// TwinCAT 3 PLC project Main
// Title: nepionic-packml
// Company: nepionic
// ProjectVersion: 0.1.0
// ProgramVersion: 3.1.4026.1+c9eadab3edd020c56c333d811d5b3c408c2550c8
// project tree:
//   Commands/ I_AbortedCommands.TcIO, I_AbortingCommands.TcIO, I_ClearingCommands.TcIO, I_CompleteCommands.TcIO, I_CompletingCommands.TcIO, I_ExecuteCommands.TcIO, I_HeldCommands.TcIO, I_HoldingCommands.TcIO, I_IdleCommands.TcIO, I_ResettingCommands.TcIO, I_StartingCommands.TcIO, I_StoppedCommands.TcIO, I_StoppingCommands.TcIO, I_SuspendedCommands.TcIO, I_SuspendingCommands.TcIO, I_UnholdingCommands.TcIO, I_UnsuspendingCommands.TcIO
//   StateMachine/ State.TcDUT, StateMachine.TcPOU
//   UnitMode/ I_UnitMode.TcIO, UnitMode.TcPOU

// ---- StateMachine/State.TcDUT
{attribute 'qualified_only'}
{attribute 'strict'}
TYPE State :
(
	UNDEFINED := 0,
    CLEARING := 1,
    STOPPED := 2,
    STARTING := 3,
    IDLE := 4,
    SUSPENDED := 5,
	EXECUTE := 6,
    STOPPING := 7,
    ABORTING := 8,
    ABORTED := 9,
    HOLDING := 10,
    HELD := 11,
    UNHOLDING := 12,
    SUSPENDING := 13,
    UNSUSPENDING := 14,
    RESETTING := 15,
    COMPLETING := 16,
    COMPLETE := 17
);
END_TYPE

// ---- Commands/I_AbortedCommands.TcIO
INTERFACE PUBLIC I_AbortedCommands

METHOD PUBLIC Clear
END_METHOD

END_INTERFACE

// ---- Commands/I_AbortingCommands.TcIO
INTERFACE PUBLIC I_AbortingCommands

METHOD PUBLIC StateComplete
END_METHOD

END_INTERFACE

// ---- Commands/I_ClearingCommands.TcIO
INTERFACE PUBLIC I_ClearingCommands

METHOD PUBLIC Abort
END_METHOD

METHOD PUBLIC StateComplete
END_METHOD

END_INTERFACE

// ---- Commands/I_CompleteCommands.TcIO
INTERFACE PUBLIC I_CompleteCommands

METHOD PUBLIC Abort
END_METHOD

METHOD PUBLIC Reset
END_METHOD

METHOD PUBLIC Stop
END_METHOD

END_INTERFACE

// ---- Commands/I_CompletingCommands.TcIO
INTERFACE PUBLIC I_CompletingCommands

METHOD PUBLIC Abort
END_METHOD

METHOD PUBLIC StateComplete
END_METHOD

METHOD PUBLIC Stop
END_METHOD

END_INTERFACE

// ---- Commands/I_ExecuteCommands.TcIO
INTERFACE PUBLIC I_ExecuteCommands

METHOD PUBLIC Abort
END_METHOD

METHOD PUBLIC Hold
END_METHOD

METHOD PUBLIC StateComplete
END_METHOD

METHOD PUBLIC Stop
END_METHOD

METHOD PUBLIC Suspend
END_METHOD

END_INTERFACE

// ---- Commands/I_HeldCommands.TcIO
INTERFACE PUBLIC I_HeldCommands

METHOD PUBLIC Abort
END_METHOD

METHOD PUBLIC Stop
END_METHOD

METHOD PUBLIC Unhold
END_METHOD

END_INTERFACE

// ---- Commands/I_HoldingCommands.TcIO
INTERFACE PUBLIC I_HoldingCommands

METHOD PUBLIC Abort
END_METHOD

METHOD PUBLIC StateComplete
END_METHOD

METHOD PUBLIC Stop
END_METHOD

END_INTERFACE

// ---- Commands/I_IdleCommands.TcIO
INTERFACE PUBLIC I_IdleCommands

METHOD PUBLIC Abort
END_METHOD

METHOD PUBLIC Start
END_METHOD

METHOD PUBLIC Stop
END_METHOD

END_INTERFACE

// ---- Commands/I_ResettingCommands.TcIO
INTERFACE PUBLIC I_ResettingCommands

METHOD PUBLIC Abort
END_METHOD

METHOD PUBLIC StateComplete
END_METHOD

METHOD PUBLIC Stop
END_METHOD

END_INTERFACE

// ---- Commands/I_StartingCommands.TcIO
INTERFACE PUBLIC I_StartingCommands

METHOD PUBLIC Abort
END_METHOD

METHOD PUBLIC StateComplete
END_METHOD

END_INTERFACE

// ---- Commands/I_StoppedCommands.TcIO
INTERFACE I_StoppedCommands

METHOD PUBLIC Reset
END_METHOD

END_INTERFACE

// ---- Commands/I_StoppingCommands.TcIO
INTERFACE PUBLIC I_StoppingCommands

METHOD PUBLIC StateComplete
END_METHOD

END_INTERFACE

// ---- Commands/I_SuspendedCommands.TcIO
INTERFACE PUBLIC I_SuspendedCommands

METHOD PUBLIC Abort
END_METHOD

METHOD PUBLIC Stop
END_METHOD

METHOD PUBLIC Unsuspend
END_METHOD

END_INTERFACE

// ---- Commands/I_SuspendingCommands.TcIO
INTERFACE PUBLIC I_SuspendingCommands

METHOD PUBLIC Abort
END_METHOD

METHOD PUBLIC StateComplete
END_METHOD

METHOD PUBLIC Stop
END_METHOD

END_INTERFACE

// ---- Commands/I_UnholdingCommands.TcIO
INTERFACE PUBLIC I_UnholdingCommands

METHOD PUBLIC Abort
END_METHOD

METHOD PUBLIC StateComplete
END_METHOD

METHOD PUBLIC Stop
END_METHOD

END_INTERFACE

// ---- Commands/I_UnsuspendingCommands.TcIO
INTERFACE PUBLIC I_UnsuspendingCommands

METHOD PUBLIC Abort
END_METHOD

METHOD PUBLIC StateComplete
END_METHOD

METHOD PUBLIC Stop
END_METHOD

END_INTERFACE

// ---- UnitMode/I_UnitMode.TcIO
INTERFACE PUBLIC I_UnitMode

METHOD PUBLIC Abort
END_METHOD

METHOD PUBLIC Clear
END_METHOD

{attribute 'monitoring':='call'}
PROPERTY PUBLIC CurrentState : State
GET
END_GET
END_PROPERTY

METHOD PUBLIC CyclicCall
END_METHOD

METHOD PUBLIC Hold
END_METHOD

{attribute 'monitoring':='call'}
PROPERTY PUBLIC IsAborted : BOOL
GET
END_GET
END_PROPERTY

{attribute 'monitoring':='call'}
PROPERTY PUBLIC IsAborting : BOOL
GET
END_GET
END_PROPERTY

{attribute 'monitoring':='call'}
PROPERTY PUBLIC IsClearing : BOOL
GET
END_GET
END_PROPERTY

{attribute 'monitoring':='call'}
PROPERTY PUBLIC IsComplete : BOOL
GET
END_GET
END_PROPERTY

{attribute 'monitoring':='call'}
PROPERTY PUBLIC IsCompleting : BOOL
GET
END_GET
END_PROPERTY

{attribute 'monitoring':='call'}
PROPERTY PUBLIC IsExecuting : BOOL
GET
END_GET
END_PROPERTY

{attribute 'monitoring':='call'}
PROPERTY PUBLIC IsHeld : BOOL
GET
END_GET
END_PROPERTY

{attribute 'monitoring':='call'}
PROPERTY PUBLIC IsHolding : BOOL
GET
END_GET
END_PROPERTY

{attribute 'monitoring':='call'}
PROPERTY PUBLIC IsIdle : BOOL
GET
END_GET
END_PROPERTY

{attribute 'monitoring':='call'}
PROPERTY PUBLIC IsResetting : BOOL
GET
END_GET
END_PROPERTY

{attribute 'monitoring':='call'}
PROPERTY PUBLIC IsStarting : BOOL
GET
END_GET
END_PROPERTY

{attribute 'monitoring':='call'}
PROPERTY PUBLIC IsStopped : BOOL
GET
END_GET
END_PROPERTY

{attribute 'monitoring':='call'}
PROPERTY PUBLIC IsStopping : BOOL
GET
END_GET
END_PROPERTY

{attribute 'monitoring':='call'}
PROPERTY PUBLIC IsSuspended : BOOL
GET
END_GET
END_PROPERTY

{attribute 'monitoring':='call'}
PROPERTY PUBLIC IsSuspending : BOOL
GET
END_GET
END_PROPERTY

{attribute 'monitoring':='call'}
PROPERTY PUBLIC IsUnholding : BOOL
GET
END_GET
END_PROPERTY

{attribute 'monitoring':='call'}
PROPERTY PUBLIC IsUnsuspending : BOOL
GET
END_GET
END_PROPERTY

METHOD PUBLIC Reset
END_METHOD

METHOD PUBLIC Start
END_METHOD

METHOD PUBLIC Stop
END_METHOD

METHOD PUBLIC Suspend
END_METHOD

METHOD PUBLIC Unhold
END_METHOD

METHOD PUBLIC Unsuspend
END_METHOD

END_INTERFACE

// ---- StateMachine/StateMachine.TcPOU
{attribute 'linkalways'} 
{attribute 'no_explicit_call' := 'This FB is a CLASS and must be accessed using methods or properties'}
{attribute 'enable_dynamic_creation'}
FUNCTION_BLOCK PUBLIC StateMachine
IMPLEMENTS
	I_AbortingCommands,
	I_ClearingCommands,
	I_HeldCommands,
	I_CompletingCommands,
	I_ExecuteCommands,
	I_AbortedCommands,
	I_CompleteCommands,
	I_HoldingCommands,
	I_UnsuspendingCommands,
	I_UnholdingCommands,
	I_SuspendingCommands,
	I_SuspendedCommands,
	I_IdleCommands,
	I_ResettingCommands,
	I_StartingCommands,
	I_StoppedCommands,
	I_StoppingCommands
VAR
	_state : State := State.IDLE;
END_VAR

METHOD PUBLIC Abort
IF IsAborting OR IsAborted THEN
	RETURN;
END_IF

_state := State.ABORTING;
END_METHOD

METHOD PUBLIC Clear
IF IsAborted THEN 
	_state := State.CLEARING;
END_IF
END_METHOD

{attribute 'monitoring':='call'}
PROPERTY PUBLIC CurrentState : State
GET
CurrentState := _state;
END_GET
END_PROPERTY

METHOD PUBLIC Hold
IF IsExecuting THEN 
	_state := State.HOLDING;
END_IF
END_METHOD

{attribute 'monitoring':='call'}
PROPERTY PUBLIC IsAborted : BOOL
GET
IsAborted := (_state = State.ABORTED);
END_GET
END_PROPERTY

{attribute 'monitoring':='call'}
PROPERTY PUBLIC IsAborting : BOOL
GET
IsAborting := (_state = State.ABORTING);
END_GET
END_PROPERTY

{attribute 'monitoring':='call'}
PROPERTY PUBLIC IsClearing : BOOL
GET
IsClearing := (_state = State.CLEARING);
END_GET
END_PROPERTY

{attribute 'monitoring':='call'}
PROPERTY PUBLIC IsComplete : BOOL
GET
IsComplete := (_state = State.COMPLETE);
END_GET
END_PROPERTY

{attribute 'monitoring':='call'}
PROPERTY PUBLIC IsCompleting : BOOL
GET
IsCompleting := (_state = State.COMPLETING);
END_GET
END_PROPERTY

{attribute 'monitoring':='call'}
PROPERTY PUBLIC IsExecuting : BOOL
GET
IsExecuting := (_state = State.EXECUTE);
END_GET
END_PROPERTY

{attribute 'monitoring':='call'}
PROPERTY PUBLIC IsHeld : BOOL
GET
IsHeld := (_state = State.HELD);
END_GET
END_PROPERTY

{attribute 'monitoring':='call'}
PROPERTY PUBLIC IsHolding : BOOL
GET
IsHolding := (_state = State.HOLDING);
END_GET
END_PROPERTY

{attribute 'monitoring':='call'}
PROPERTY PUBLIC IsIdle : BOOL
GET
isIdle := (_state = State.IDLE);
END_GET
END_PROPERTY

{attribute 'monitoring':='call'}
PROPERTY PUBLIC IsResetting : BOOL
GET
IsResetting := (_state = State.RESETTING);
END_GET
END_PROPERTY

{attribute 'monitoring':='call'}
PROPERTY PUBLIC IsStarting : BOOL
GET
IsStarting := (_state = State.STARTING);
END_GET
END_PROPERTY

{attribute 'monitoring':='call'}
PROPERTY PUBLIC IsStopped : BOOL
GET
isStopped := (_state = State.STOPPED);
END_GET
END_PROPERTY

{attribute 'monitoring':='call'}
PROPERTY PUBLIC IsStopping : BOOL
GET
IsStopping := (_state = State.STOPPING);
END_GET
END_PROPERTY

{attribute 'monitoring':='call'}
PROPERTY PUBLIC IsSuspended : BOOL
GET
IsSuspended := (_state = State.SUSPENDED);
END_GET
END_PROPERTY

{attribute 'monitoring':='call'}
PROPERTY PUBLIC IsSuspending : BOOL
GET
IsSuspending := (_state = State.SUSPENDING);
END_GET
END_PROPERTY

{attribute 'monitoring':='call'}
PROPERTY PUBLIC IsUnholding : BOOL
GET
IsUnholding := (_state = State.UNHOLDING);
END_GET
END_PROPERTY

{attribute 'monitoring':='call'}
PROPERTY PUBLIC IsUnsuspending : BOOL
GET
IsUnsuspending := (_state = State.UNSUSPENDING);
END_GET
END_PROPERTY

METHOD PUBLIC Reset
IF IsStopped OR IsComplete THEN 
	_state := State.RESETTING;
END_IF
END_METHOD

METHOD PUBLIC Start
IF IsIdle THEN 
	_state := State.STARTING;
END_IF
END_METHOD

METHOD PUBLIC StateComplete
CASE _state OF 
	State.IDLE : RETURN;
	State.STARTING : _state := State.EXECUTE;
	State.EXECUTE : _state := State.COMPLETING;
	State.COMPLETING : _state := State.COMPLETE;
	State.COMPLETE : RETURN;
	State.STOPPING : _state := State.STOPPED;
	State.STOPPED : RETURN;
	State.RESETTING : _state := State.IDLE;
	State.HOLDING : _state := State.HELD;
	State.HELD : RETURN;
	State.UNHOLDING : _state := State.EXECUTE;
	State.SUSPENDING : _state := State.SUSPENDED;
	State.SUSPENDED : RETURN;
	State.UNSUSPENDING : _state := State.EXECUTE;
	State.CLEARING : _state := State.STOPPED;
	State.ABORTED : RETURN;
	State.ABORTING : _state := State.ABORTED;
END_CASE
END_METHOD

METHOD PUBLIC Stop
CASE _state OF
	State.STOPPED: RETURN;
	State.STOPPING: RETURN;
	State.CLEARING: RETURN;
	State.ABORTED: RETURN;
	State.ABORTING: RETURN;
END_CASE

_state := State.STOPPING;
END_METHOD

METHOD PUBLIC Suspend
IF IsExecuting THEN 
	_state := State.SUSPENDING;
END_IF
END_METHOD

METHOD PUBLIC Unhold
IF IsHeld THEN 
	_state := State.UNHOLDING;
END_IF
END_METHOD

METHOD PUBLIC Unsuspend
IF IsSuspended THEN 
	_state := State.UNSUSPENDING;
END_IF
END_METHOD

END_FUNCTION_BLOCK

// ---- UnitMode/UnitMode.TcPOU
{attribute 'linkalways'} 
{attribute 'no_explicit_call' := 'This FB is a CLASS and must be accessed using methods or properties'}
{attribute 'enable_dynamic_creation'}
FUNCTION_BLOCK PUBLIC ABSTRACT UnitMode IMPLEMENTS I_UnitMode
VAR
	stateMachine : StateMachine;
END_VAR

METHOD PUBLIC Abort
stateMachine.Abort();
END_METHOD

METHOD PROTECTED Aborted
VAR_INPUT
	commands : I_AbortedCommands;
END_VAR
END_METHOD

METHOD PROTECTED Aborting
VAR_INPUT
	commands : I_AbortingCommands;
END_VAR
commands.StateComplete();
END_METHOD

METHOD PUBLIC Clear
stateMachine.Clear();
END_METHOD

METHOD PROTECTED Clearing
VAR_INPUT
	commands : I_ClearingCommands;
END_VAR
commands.StateComplete();
END_METHOD

METHOD PROTECTED Complete
VAR_INPUT
	commands : I_CompleteCommands;
END_VAR
END_METHOD

METHOD PROTECTED Completing
VAR_INPUT
	commands : I_CompletingCommands;
END_VAR
commands.StateComplete();
END_METHOD

{attribute 'monitoring':='call'}
PROPERTY PUBLIC CurrentState : State
GET
CurrentState := stateMachine.CurrentState;
END_GET
END_PROPERTY

METHOD PUBLIC CyclicCall
IF stateMachine.IsIdle THEN 
	Idle(stateMachine);
END_IF

IF stateMachine.IsStarting THEN
	Starting(stateMachine);
END_IF

IF stateMachine.IsExecuting THEN
	Execute(stateMachine);
END_IF

IF stateMachine.IsCompleting THEN
	Completing(stateMachine);
END_IF

IF stateMachine.IsComplete THEN
	Complete(stateMachine);
END_IF

IF stateMachine.IsStopping THEN
	Stopping(stateMachine);
END_IF

IF stateMachine.IsStopped THEN
	Stopped(stateMachine);
END_IF

IF stateMachine.IsResetting THEN
	Resetting(stateMachine);
END_IF

IF stateMachine.IsHolding THEN
	Holding(stateMachine);
END_IF

IF stateMachine.IsHeld THEN
	Held(stateMachine);
END_IF

IF stateMachine.IsUnholding THEN
	Unholding(stateMachine);
END_IF

IF stateMachine.IsSuspending THEN
	Suspending(stateMachine);
END_IF

IF stateMachine.IsSuspended THEN
	Suspended(stateMachine);
END_IF

IF stateMachine.IsUnsuspending THEN
	Unsuspending(stateMachine);
END_IF

IF stateMachine.IsClearing THEN
	Clearing(stateMachine);
END_IF

IF stateMachine.IsAborted THEN
	Aborted(stateMachine);
END_IF

IF stateMachine.IsAborting THEN
	Aborting(stateMachine);
END_IF
END_METHOD

METHOD PROTECTED Execute
VAR_INPUT
	commands : I_ExecuteCommands;
END_VAR
commands.StateComplete();
END_METHOD

METHOD PROTECTED Held
VAR_INPUT
	commands : I_HeldCommands;
END_VAR
END_METHOD

METHOD PUBLIC Hold
stateMachine.Hold();
END_METHOD

METHOD PROTECTED Holding
VAR_INPUT
	commands : I_HoldingCommands;
END_VAR
commands.StateComplete();
END_METHOD

METHOD PROTECTED Idle
VAR_INPUT
	commands : I_IdleCommands;
END_VAR
END_METHOD

{attribute 'monitoring':='call'}
PROPERTY PUBLIC IsAborted : bool
GET
IsAborted := stateMachine.IsAborted;
END_GET
END_PROPERTY

{attribute 'monitoring':='call'}
PROPERTY PUBLIC IsAborting : bool
GET
IsAborting := stateMachine.IsAborting;
END_GET
END_PROPERTY

{attribute 'monitoring':='call'}
PROPERTY PUBLIC IsClearing : bool
GET
IsClearing := stateMachine.IsClearing;
END_GET
END_PROPERTY

{attribute 'monitoring':='call'}
PROPERTY PUBLIC IsComplete : bool
GET
IsComplete := stateMachine.IsComplete;
END_GET
END_PROPERTY

{attribute 'monitoring':='call'}
PROPERTY PUBLIC IsCompleting : bool
GET
IsCompleting := stateMachine.IsCompleting;
END_GET
END_PROPERTY

{attribute 'monitoring':='call'}
PROPERTY PUBLIC IsExecuting : bool
GET
IsExecuting := stateMachine.IsExecuting;
END_GET
END_PROPERTY

{attribute 'monitoring':='call'}
PROPERTY PUBLIC IsHeld : bool
GET
IsHeld := stateMachine.IsHeld;
END_GET
END_PROPERTY

{attribute 'monitoring':='call'}
PROPERTY PUBLIC IsHolding : bool
GET
IsHolding := stateMachine.IsHolding;
END_GET
END_PROPERTY

{attribute 'monitoring':='call'}
PROPERTY PUBLIC IsIdle : BOOL
GET
isIdle := stateMachine.isIdle;
END_GET
END_PROPERTY

{attribute 'monitoring':='call'}
PROPERTY PUBLIC IsResetting : bool
GET
IsResetting := stateMachine.IsResetting;
END_GET
END_PROPERTY

{attribute 'monitoring':='call'}
PROPERTY PUBLIC IsStarting : bool
GET
IsStarting := stateMachine.IsStarting;
END_GET
END_PROPERTY

{attribute 'monitoring':='call'}
PROPERTY PUBLIC IsStopped : BOOL
GET
isStopped := stateMachine.isStopped;
END_GET
END_PROPERTY

{attribute 'monitoring':='call'}
PROPERTY PUBLIC IsStopping : bool
GET
IsStopping := stateMachine.IsStopping;
END_GET
END_PROPERTY

{attribute 'monitoring':='call'}
PROPERTY PUBLIC IsSuspended : bool
GET
IsSuspended := stateMachine.IsSuspended;
END_GET
END_PROPERTY

{attribute 'monitoring':='call'}
PROPERTY PUBLIC IsSuspending : bool
GET
IsSuspending := stateMachine.IsSuspending;
END_GET
END_PROPERTY

{attribute 'monitoring':='call'}
PROPERTY PUBLIC IsUnholding : bool
GET
IsUnholding := stateMachine.IsUnholding;
END_GET
END_PROPERTY

{attribute 'monitoring':='call'}
PROPERTY PUBLIC IsUnsuspending : bool
GET
IsUnsuspending := stateMachine.IsUnsuspending;
END_GET
END_PROPERTY

METHOD PUBLIC Reset
stateMachine.Reset();
END_METHOD

METHOD PROTECTED Resetting
VAR_INPUT
	commands : I_ResettingCommands;
END_VAR
commands.StateComplete();
END_METHOD

METHOD PUBLIC Start
stateMachine.Start();
END_METHOD

METHOD PROTECTED Starting
VAR_INPUT
	commands : I_StartingCommands;
END_VAR
commands.StateComplete();
END_METHOD

METHOD PUBLIC Stop
stateMachine.Stop();
END_METHOD

METHOD PROTECTED Stopped
VAR_INPUT
	commands : I_StoppedCommands;
END_VAR
END_METHOD

METHOD PROTECTED Stopping
VAR_INPUT
	commands : I_StoppingCommands;
END_VAR
commands.StateComplete();
END_METHOD

METHOD PUBLIC Suspend
stateMachine.Suspend();
END_METHOD

METHOD PROTECTED Suspended
VAR_INPUT
	commands : I_SuspendedCommands;
END_VAR
END_METHOD

METHOD PROTECTED Suspending
VAR_INPUT
	commands : I_SuspendingCommands;
END_VAR
commands.StateComplete();
END_METHOD

METHOD PUBLIC Unhold
stateMachine.Unhold();
END_METHOD

METHOD PROTECTED Unholding
VAR_INPUT
	commands : I_UnholdingCommands;
END_VAR
commands.StateComplete();
END_METHOD

METHOD PUBLIC Unsuspend
stateMachine.Unsuspend();
END_METHOD

METHOD PROTECTED Unsuspending
VAR_INPUT
	commands : I_UnsuspendingCommands;
END_VAR
commands.StateComplete();
END_METHOD

END_FUNCTION_BLOCK
